Staubli VAL3: setAllSpeed.pgx

program setAllSpeed(num x_nNewValue (dimensions=1), num x_nOldValue (dimensions=1))
  local num i
  local num l_nSize
  local TrajectoryItem l_tTraj
begin
  // change all the speed
  if x_nNewValue!=x_nOldValue
    call trajType:getSizeItem(false,l_nSize)
    // scan it
    for i=0 to (l_nSize-1)
      // get the trajitem
      call trajType:getTrajItem(l_tTraj,i)
      // JOINT MOVEMENT
      if (l_tTraj.moveType==0) and (x_nOldValue==l_tTraj.nom_speed.vel)
        l_tTraj.nom_speed.vel=x_nNewValue
        // LINEAR MOVEMENT
      elseIf (l_tTraj.moveType==1 or l_tTraj.moveType==2) and (x_nOldValue==l_tTraj.nom_speed.tvel)
        l_tTraj.nom_speed.tvel=x_nNewValue
      endIf
      // set the trajItem
      call trajType:setTrajItem(l_tTraj,i)
    endFor
  endIf
end
